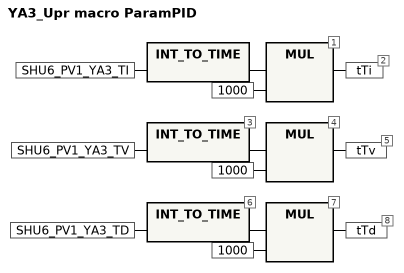
[picture p440: YA3_Upr macro ParamPID (CFC)]
_CFC_ (* Continuous Function Chart, elements in execution order *)
#0 SHU6_YA3_REQ_VYHOD <= #49
#1 TON_SHU6_PV1_P1_DI5_RUN:TON(IN: SHU6_PV1_1P1_DI4_RUN, PT: T#10s)
#2 AND(SHU6_PV1_UST_RE_RABOTA, #1.Q)
#3 reg1 <= #2
#4 AND(NOT SHU6_PV1_UST_RE_RABOTA, #1.Q, NOT SHU6_PV1_UST_RE_PROGREV)
#5 reg2 <= #4
#6 MACRO ParamPID()
	#7 INT_TO_TIME(SHU6_PV1_YA3_TI)
	#8 MUL(#7, 1000)
	#9 tTi <= #8
	#10 INT_TO_TIME(SHU6_PV1_YA3_TV)
	#11 MUL(#10, 1000)
	#12 tTv <= #11
	#13 INT_TO_TIME(SHU6_PV1_YA3_TD)
	#14 MUL(#13, 1000)
	#15 tTd <= #14
END_MACRO
#16 SUB(SHU6_PV1_TE6_UST, SHU6_PV1_TE4_VN)
#17 EPS2 <= #16
#18 AND(reg1, SHU6_PV1_TE6_DOST)
#19 AND(reg2, SHU6_PV1_TE4_DOST)
#20 OR(#18, #19)
#21 YA3_DOST <= #20
#22 SUB(SHU6_PV1_TE6_UST, SHU6_PV1_TE6_VN)
#23 EPS1 <= #22
#24 YA3_AVT <= #38
#25 SEL(reg1, SHU6_PV1_TE4_UST, SHU6_PV1_TE6_UST)
#26 >(EPS1, EPS2)
#27 AND(reg1, #26)
#28 SEL(#27, SHU6_PV1_TE4_VN, SHU6_PV1_TE6_VN)
#29 OR(reg1, reg2)
#30 AND(#29, YA3_DOST)
#31 SEL(#30, 0, #25)
#32 SEL(#30, 0, #28)
#33 AND(#30, SHU6_PV1_1YA3_DI1_A)
#34 SHU6_PV1_YA3_AUTO <= #33
#35 AND(NOT SHU6_PV1_TE1_B_UST_MYAG_REG, SHU6_PV1_UST_RE_PROGREV)
#36 OR(Z_ZAM_SR, #35)
#37 AND(#33, NOT #36)
#38 AND(#37, NOT SHU6_PV1_Z_GVS1_OTKAZ)
#39 YA3_REG_POL <= #38
#40 SEL(#38, eHVACCtrlMode_Manual, eHVACCtrlMode_Auto)
#41 SEL(NOT SHU6_PV1_1P1_DI4_RUN, SHU6_PV1_YA3_UP_VN, rYMin)
#42 SEL(SHU6_PV1_UST_RE_PROGREV, #41, 50)
#43 SEL(#36, #42, 100)
#44 SEL(SHU6_PV1_1YA3_DI1_A, SHU6_PV1_YA3_UP_VN, #43)
#45 SEL(SHU6_PV1_Z_GVS1_OTKAZ, #44, 0)
#46 YA3_PID:FB_HVACPIDCtrl(eHVACDataSecurityType_Idle, FALSE, TRUE, #31, #32, tTaskCycleTime, tTaskCycleTime, #40, #45, SHU6_PV1_YA3_UP_VN, FALSE, SHU6_PV1_SB, deadRange, direction, SHU6_PV1_YA3_KP, tTi, tTv, tTd, rYMin, rYMax)
#47 SHU6_PV1_YA3_RASSOG <= #46.out 2
#48 YA3_OTKAZ <= #46.out 8
#49 SEL(SHU6_PV1_1YA3_DI1_A, 0, #46.out 1)
#50 SUB(#49, SHU6_PV1_YA3_UP_VN)
#51 SHU6_PV1_YA3_RASSOG_POL <= #50
#52 SEL(SHU6_PV1_UST_ZIMA, 0, SHU6_PV1_YA3_UP_MIN)
#53 rYMin <= #52
_END_CFC_
END_PROGRAM

(* POU IM/YA4_Upr, CFC *)
PROGRAM YA4_Upr
VAR
	YA3_PID: FB_HVACPIDCtrl;

	deadRange: REAL := 0.1;
	direction: BOOL := TRUE;
	tTi: TIME;
	tTv: TIME;
	tTd: TIME;

	rYMin: REAL := 0;
	rYMax: REAL := 100;
END_VAR
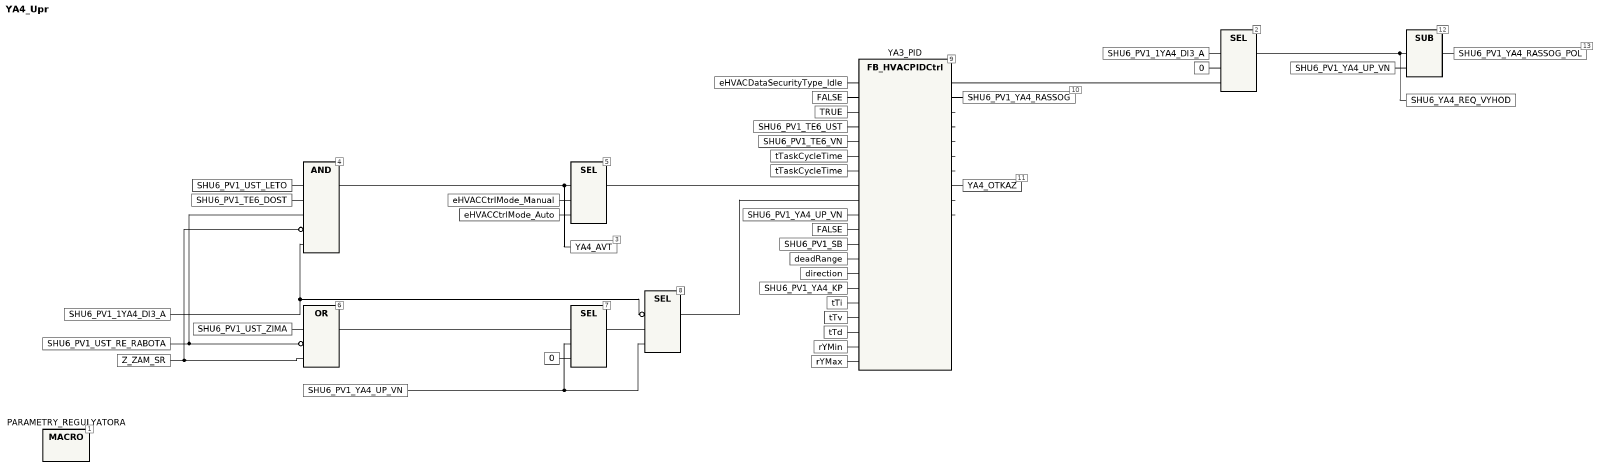
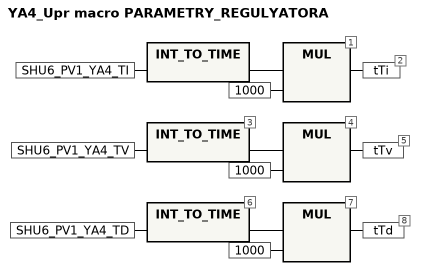
_CFC_ (* Continuous Function Chart, elements in execution order *)
#0 SHU6_YA4_REQ_VYHOD <= #11
#1 MACRO PARAMETRY_REGULYATORA()
	#2 INT_TO_TIME(SHU6_PV1_YA4_TI)
	#3 MUL(#2, 1000)
	#4 tTi <= #3
	#5 INT_TO_TIME(SHU6_PV1_YA4_TV)
	#6 MUL(#5, 1000)
	#7 tTv <= #6
	#8 INT_TO_TIME(SHU6_PV1_YA4_TD)
	#9 MUL(#8, 1000)
	#10 tTd <= #9
END_MACRO
#11 SEL(SHU6_PV1_1YA4_DI3_A, 0, #18.out 1)
#12 YA4_AVT <= #13
#13 AND(SHU6_PV1_UST_LETO, SHU6_PV1_TE6_DOST, SHU6_PV1_UST_RE_RABOTA, NOT Z_ZAM_SR, SHU6_PV1_1YA4_DI3_A)
#14 SEL(#13, eHVACCtrlMode_Manual, eHVACCtrlMode_Auto)
#15 OR(SHU6_PV1_UST_ZIMA, NOT SHU6_PV1_UST_RE_RABOTA, Z_ZAM_SR)
#16 SEL(#15, SHU6_PV1_YA4_UP_VN, 0)
#17 SEL(NOT SHU6_PV1_1YA4_DI3_A, #16, SHU6_PV1_YA4_UP_VN)
#18 YA3_PID:FB_HVACPIDCtrl(eHVACDataSecurityType_Idle, FALSE, TRUE, SHU6_PV1_TE6_UST, SHU6_PV1_TE6_VN, tTaskCycleTime, tTaskCycleTime, #14, #17, SHU6_PV1_YA4_UP_VN, FALSE, SHU6_PV1_SB, deadRange, direction, SHU6_PV1_YA4_KP, tTi, tTv, tTd, rYMin, rYMax)
#19 SHU6_PV1_YA4_RASSOG <= #18.out 2
#20 YA4_OTKAZ <= #18.out 8
#21 SUB(#11, SHU6_PV1_YA4_UP_VN)
#22 SHU6_PV1_YA4_RASSOG_POL <= #21
_END_CFC_
END_PROGRAM

(* POU IM/razr_pusk, CFC *)
PROGRAM razr_pusk
VAR
END_VAR
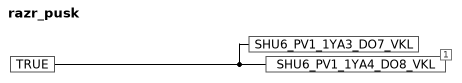
_CFC_ (* Continuous Function Chart, elements in execution order *)
#0 SHU6_PV1_1YA3_DO7_VKL <= TRUE
#1 SHU6_PV1_1YA4_DO8_VKL <= TRUE
_END_CFC_
(* the same logic as Structured Text *)
SHU6_PV1_1YA3_DO7_VKL := TRUE;
SHU6_PV1_1YA4_DO8_VKL := TRUE;
END_PROGRAM

(* POU IM/BLOK_SINH_DVUH_REG, CFC *)
PROGRAM BLOK_SINH_DVUH_REG
VAR
	res_1: REAL;
	res_2: BOOL;
	res_3: BOOL;
	res_4: BOOL;

	RS_BLOKIROVKA: RS;
	RS_UST_BLOK: R_TRIG;
	RS_SB_BLOK: R_TRIG;
END_VAR
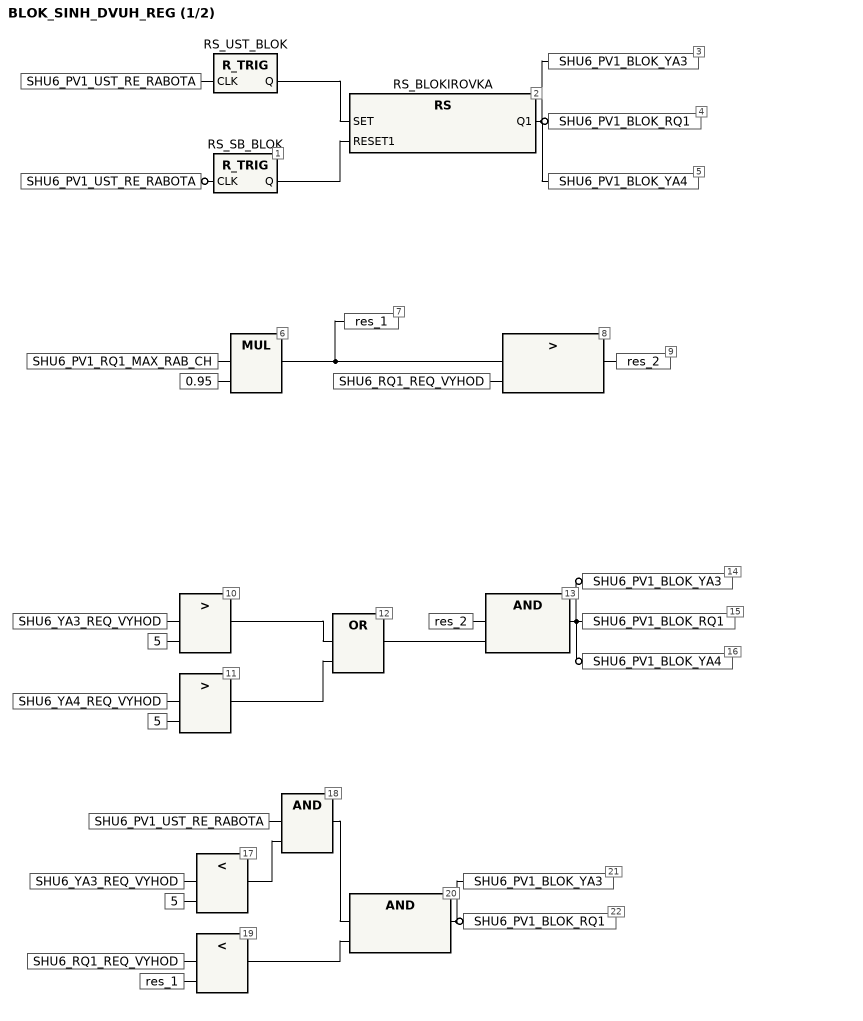
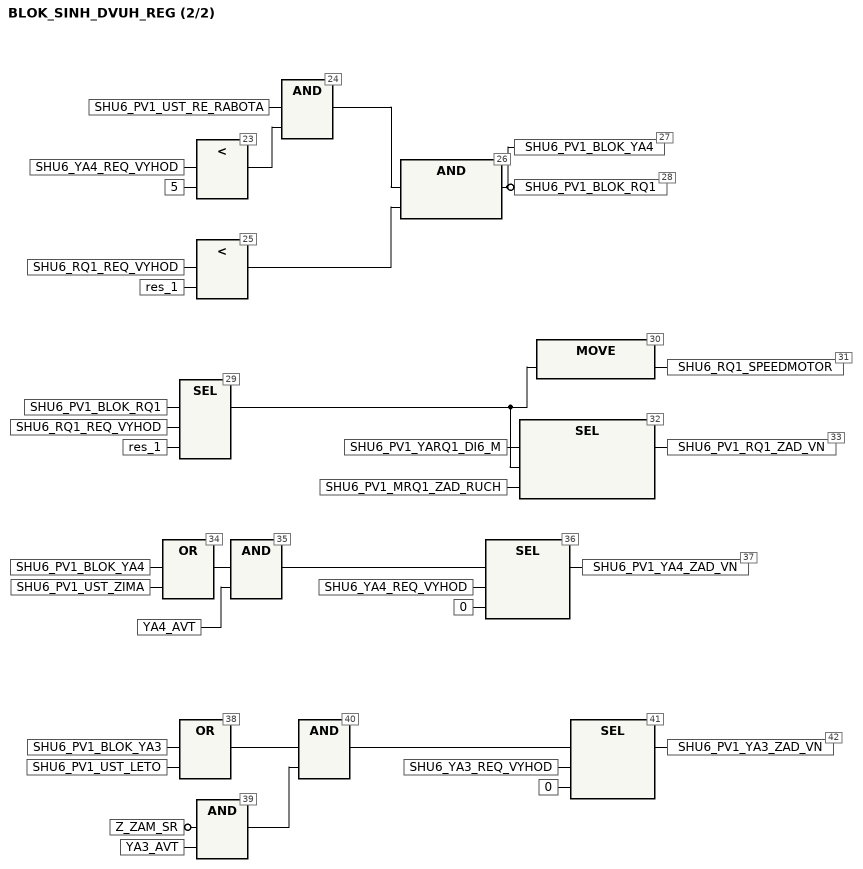
